// Startup hook called after PreInit and before PostInit.
INTERFACE I_Init EXTENDS I_Generic

// Called once during Plant startup.
METHOD Init
END_METHOD

END_INTERFACE

(* stored: Version 1.1.0.1
   Itf I_Init: Id {4a2c0968-9644-42ff-9859-1d46f6462d6d}
   Method Init: Id {91c58654-3ffc-4818-95da-e43400094954} *)
